// TIA Portal V16 export
// export: Created 2022-11-17T11:55:30.12265Z, ExportSetting WithDefaults, DisplayName Totally Integrated Automation Portal, DisplayVersion V16 Update 6, DisplayName TIA Portal Version Control Interface, DisplayVersion V16 Update 2, DisplayName TIA Portal Openness, DisplayVersion V16 Update 6, DisplayName SINAMICS Startdrive Advanced, DisplayVersion V16 Update 5, DisplayName SINAMICS Startdrive G130, G150, S120, S150, SINAMICS MV, S210, DisplayVersion V16 Update 5, DisplayName SINAMICS Startdrive G110M, G120, G120C, G120D, G120P, G115D, DisplayVersion V16 Update 5, DisplayName STEP 7 Professional, DisplayVersion V16 Update 6, DisplayName STEP 7 Safety, DisplayVersion V16, DisplayName WinCC Advanced, DisplayVersion V16 Update 6
DATA_BLOCK "DB88_Top"   // DB88
{ S7_Optimized_Access := 'FALSE' }
AUTHOR : Robopac
VERSION : 0.0
// stored: AutoNumber false, IsOnlyStoredInLoadMemory false, IsWriteProtectedInAS false
   VAR RETAIN
      VW800 : Int := 0;
      VW802 : Int := 0;
      V804_0 : Bool := FALSE;   // Top carriage in cut position
      V804_1 : Bool := FALSE;   // Top carriage in forward position
      V804_2 : Bool := FALSE;
      V804_3 : Bool := FALSE;   // Memory to stop top carriage forward in manual mode
      V804_4 : Bool := FALSE;   // Memory for top cut done
      V804_5 : Bool := FALSE;
      V804_6 : Bool := FALSE;
      V804_7 : Bool := FALSE;
      VB805 : Byte := 16#00;
      VW806 : Int := 0;   // Top positioning counter
   END_VAR
BEGIN
END_DATA_BLOCK
